RoboDK station: robotik-project-wise24.rdk

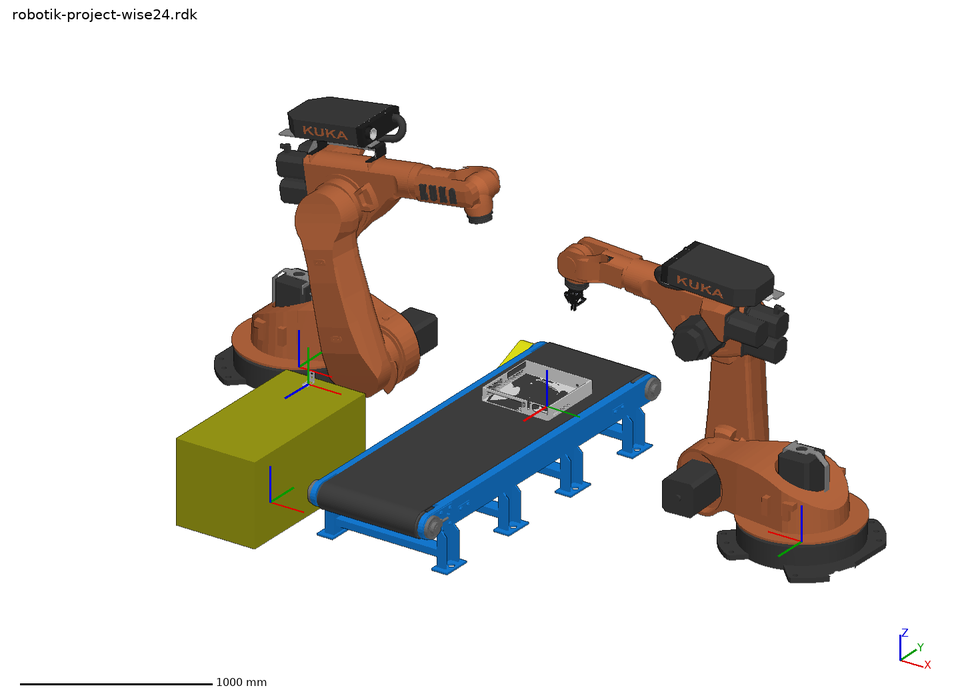
[picture v0: the station drawn from its stored meshes, robots at their saved joint values, targets as dots, program paths as lines]
Station robotik-project-wise24 (saved by RoboDK 5.8.0). Poses are relative to the parent item; angles as X-Y-Z fixed-axis rotations.
Station parameters (name, value as stored): LIN64
  - frame Conveyor Belt Wide (2m) Base at (1325.37, 352.24, 0) mm, rotated rx 0 ry 0 rz -90 deg
    - robot Conveyor Belt Wide (2m): 1 axes
        modified DH rows (alpha deg, a mm, theta deg, d mm): 0, 0, 0, 0 linear
        base shift (0, 0, 0) mm, rotated rx 0 ry 90 rz 0 deg
        joint limits [-900000] to [900000]; home [0]; saved at [0]
  - object Geha at (1650, -200, 366.5) mm, rotated rx 90 ry 0 rz 0 deg, size 420 x 80 x 400 mm, geometry from use v4.stl
  - frame KUKA KR 60 4 KS Base at (3326.41, -200, 0) mm, rotated rx 0 ry 0 rz 180 deg
    - robot KUKA KR 60 4 KS: 6 axes, payload 60 kg, reach 2233 mm, repeatability 0.06 mm, weight 600 kg
        modified DH rows (alpha deg, a mm, theta deg, d mm): 0, 0, 0, 250; -90, 550, 0, 0; 0, 850, -90, 0; -90, 145, 0, 820; 90, 0, 0, 0; -90, 0, 180, 170
        joint limits [-150, -105, -120, -350, -119, -350] to [150, 75, 158, 350, 119, 350]; home [0, -90, 90, 0, 0, 0]; saved at [-3.424, -90.58, 86.403, 0.992, 86.004, 3.241]
      - tool RobotiQ 2F-85 Gripper (Fully Closed), TCP at (0, 0, 130) mm, size 121.5 x 75 x 160.2 mm
  - frame KUKA KR 60 4 KS Base at (0, 0, 0) mm
    - robot KUKA KR 60 4 KS: 6 axes, payload 60 kg, reach 2233 mm, repeatability 0.06 mm, weight 600 kg
        modified DH rows (alpha deg, a mm, theta deg, d mm): 0, 0, 0, 250; -90, 550, 0, 0; 0, 850, -90, 0; -90, 145, 0, 820; 90, 0, 0, 0; -90, 0, 180, 170
        joint limits [-150, -105, -120, -350, -119, -350] to [150, 75, 158, 350, 119, 350]; home [0, -90, 90, 0, 0, 0]; saved at [0, -104.818, 95.943, 0, 88.571, 0]
  - frame Frame 4 at (800, -1400, 0) mm
    - object Prism 1000x500x500mm at (0, 0, 0) mm, size 500 x 1000 x 500 mm, geometry from Prism-1000x500x500mm.sld
    - frame Frame 5 at (-55.2, 420.66, 500) mm, rotated rx 90 ry 0 rz 0 deg
      - object Montagewinkel v1 at (0, 0, 0) mm, size 40 x 65 x 65 mm, geometry from Montagewinkel v1.stl
